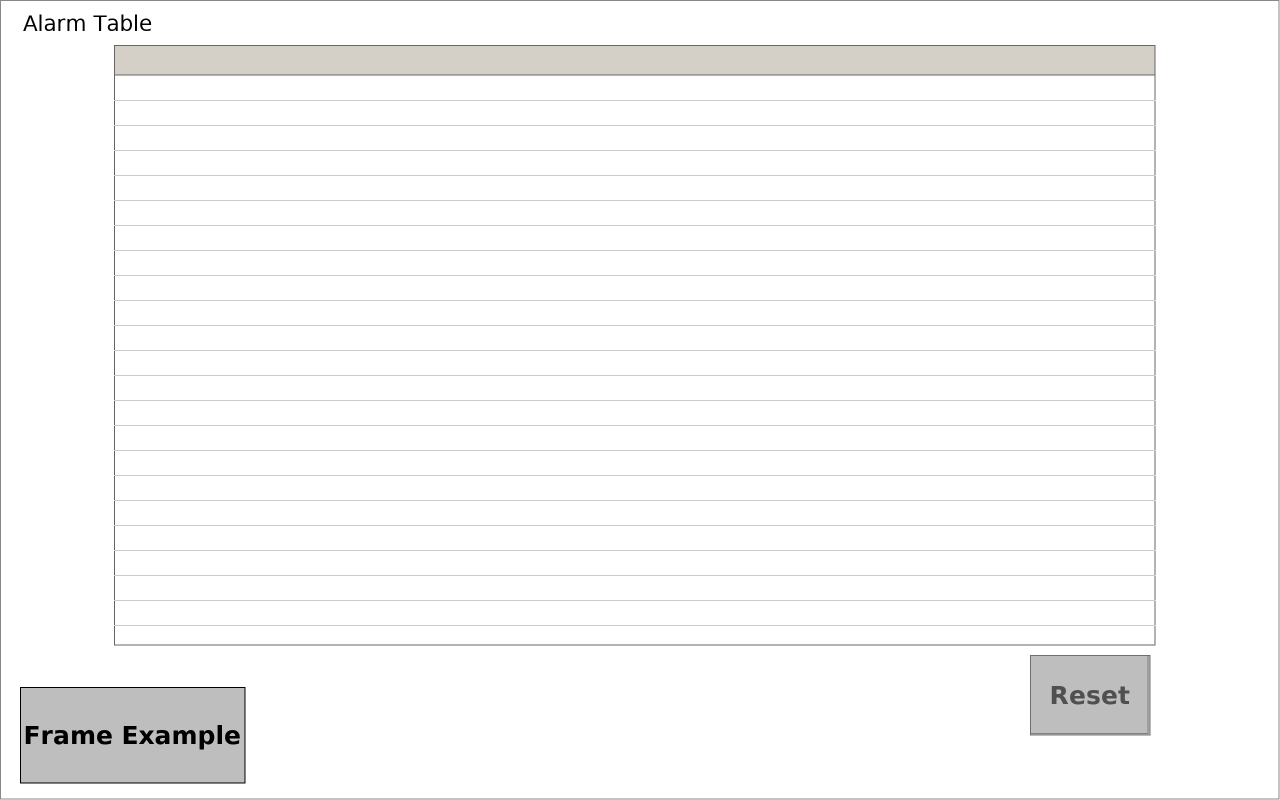
VISUALIZATION Alarm_Table  // 1280x800
    Rectangle (20,9 909x60), "Alarm Table"
    Table (114,45 1041x600), text list: 'Alarm_TextList', data array: HMI.astActiveAlarmsTable
        p1014161805: 50 - 1 + INT#1
        p3854506369: HMI.astActiveAlarmsTable[INDEX].qActive
        p1892666644: HMI.astActiveAlarmsTable[INDEX].diEventID
        p338671338: HMI.astActiveAlarmsTable[INDEX].iClass
        p2170511999: HMI.astActiveAlarmsTable[INDEX].sTime
        p3723444502: HMI.astActiveAlarmsTable[INDEX].sEvent
    Rectangle (20,687 225x96), "Frame Example"
        OnMouseClick: change screen: Alarms
    Button (1030,655 120x80), "Reset"
        tap HMI.xFaultResetPB
END_VISUALIZATION

(* stored: Version 1.1.0.1
   Visu Alarm_Table: Id {3c645d3a-d9e7-4fb0-af6f-bef3c831edf9} *)
